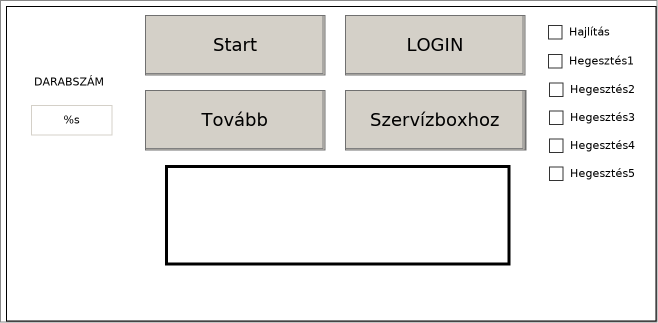
VISUALIZATION Termeles1  // 658x323
    Rectangle (6,6 650x315)
    Button (145,15 180x60), "Start"
        OnMouseUp: execute { AUTOMATA.iState:=1; }
    Button (145,90 180x60), "Tovább"
        OnMouseUp: execute { AUTOMATA.bContinue:=TRUE; }
    Button (346,90 180x60), "STOP"
        OnMouseUp: execute {
            AUTOMATA.bContinue:=FALSE;
            AUTOMATA.iState:=0;
            AUTOMATA.bWelderReservedBy1:=FALSE;
            AUTOMATA.bRobotReservedBy1:=FALSE;
        }
    Button (345,90 180x60), "Szervízboxhoz"
        OnMouseUp: execute { AUTOMATA.iState:=100; }
    Textfield (31,105 81x30), "%s", text variable: GVL.nProductCount1, input disabled if: TRUE
    Label (28,67 82x30), "DARABSZÁM"
    Checkbox (546,17 105x30), "Hajlítás", variable: GVL.bHajlitasBe, input disabled if: AUTOMATA.bFolyamatBeallitas1Tiltva
    Checkbox (546,46 105x30), "Hegesztés1", variable: GVL.bHegesztes1Be, input disabled if: AUTOMATA.bFolyamatBeallitas1Tiltva
    Checkbox (547,75 105x29), "Hegesztés2", variable: GVL.bHegesztes2Be, input disabled if: AUTOMATA.bFolyamatBeallitas1Tiltva
    Checkbox (547,103 105x29), "Hegesztés3", variable: GVL.bHegesztes3Be, input disabled if: AUTOMATA.bFolyamatBeallitas1Tiltva
    Checkbox (547,131 105x29), "Hegesztés4", variable: GVL.bHegesztes4Be, input disabled if: AUTOMATA.bFolyamatBeallitas1Tiltva
    Checkbox (547,159 105x29), "Hegesztés5", variable: GVL.bHegesztes5Be, input disabled if: AUTOMATA.bFolyamatBeallitas1Tiltva
    Button (345,15 180x60), "LOGIN"
        OnMouseClick: VisuUserMgmt Type=Login
    RoundedRectangle (235,190 215x50), text list: 'ErrorList1', text index: AUTOMATA.iState
    Label (265,160 145x30), "JELENLEGI FOLYAMAT:"
    RoundedRectangle (165,165 345x100), text list: 'ErrorList1', text index: AUTOMATA.iState
END_VISUALIZATION

(* stored: Version 1.1.0.1, ProductVersion 3.1.4024.11
   Visu Termeles1: Id {b798ec64-d9fe-41ca-b9ae-dc127305755f} *)
